FUNCTION Convert_TIME_TO_USINT : Hresult
VAR_INPUT
	in : TIME;
	out : REFERENCE TO USINT;
END_VAR
VAR
	converted : USINT;
END_VAR

converted := TIME_TO_USINT(in);

IF (USINT_TO_TIME(converted) <> in) THEN
	Convert_TIME_TO_USINT := INCOMPATIBLE;
	RETURN;
END_IF

out := converted;

END_FUNCTION

(* stored: Version 1.1.0.1, ProductVersion 3.1.4024.12
   POU Convert_TIME_TO_USINT: Id {5cd5ba8f-b26f-49c9-a077-c0c0ae8f0d66}, SpecialFunc None *)
